// TIA Portal project "Quizshow" (V20)

(* hardware
DEVICE "S7-300/ET200M-Station_1"  S7-300 station
   slot 0: "Profilschiene_0"  Rail  6ES7 390-1***0-0AA0
   slot 2: "PLC_1"  CPU 315-2 PN/DP  6ES7 315-2EH14-0AB0  V3.2.18
      slot 2: "PROFINET-Schnittstelle_1"  PN-IO
         slot 1: "Port_1"  Port
         slot 2: "Port_2"  Port
   slot 4: "DI 16x24VDC_1"  DI16 x 24VDC, interrupt  6ES7 321-7BH01-0AB0
   slot 5: "DO 8x24VDC/0.5A_1"  DO8 x 24VDC / 0.5A  6ES7 322-8BF00-0AB0
*)

// ===== PLC "PLC_1"  CPU 315-2 PN/DP =====

VAR_GLOBAL   // PLC tag table "Standard-Variablentabelle"
   "Teilnehmer_1" AT %E0.0 : Bool;
   "Teilnehmer_2" AT %E0.1 : Bool;
   "TN_1-Lampe" AT %A0.0 : Bool;
   "TN_2-Lampe" AT %A0.1 : Bool;
   "TN_2-Gedrückt" AT %M0.1 : Bool;
   "TN_1-Gedrückt" AT %M0.0 : Bool;
   "Start-Taster" AT %E1.0 : Bool;
   "Freigabe erteilt" AT %A0.7 : Bool;
   "TN_3-Lampe" AT %A0.2 : Bool;
   "TN_4-Lampe" AT %A0.3 : Bool;
   "Teilnehmer_3" AT %E0.2 : Bool;
   "Teilnehmer_4" AT %E0.3 : Bool;
   "TN_3-Gedrückt" AT %M0.2 : Bool;
   "TN_4-Gedrückt" AT %M0.3 : Bool;
END_VAR

DATA_BLOCK "Quizshow_DB"   // DB1
{ S7_Optimized_Access := 'FALSE' }
VERSION : 0.1
// stored: InstanceOfName Quizshow
"Quizshow"
BEGIN
END_DATA_BLOCK

FUNCTION_BLOCK "Quizshow"   // FB6, FBD
{ S7_Optimized_Access := 'FALSE' }
VERSION : 0.1
BEGIN

REGION Network 1: Buzzer-Teilnehmer 1
   // Siehe Netzwerk 4.
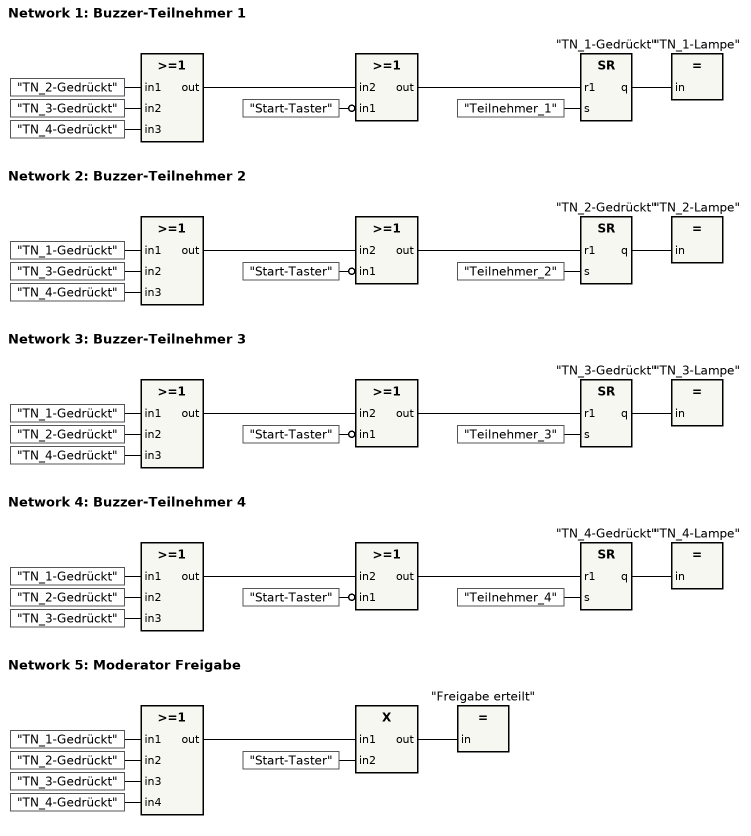
   IF "Teilnehmer_1" THEN
       "TN_1-Gedrückt" := TRUE;   // SR flip-flop
   END_IF;
   IF "TN_2-Gedrückt" OR "TN_3-Gedrückt" OR "TN_4-Gedrückt" OR NOT "Start-Taster" THEN
       "TN_1-Gedrückt" := FALSE;
   END_IF;
   "TN_1-Lampe" := "TN_1-Gedrückt";
END_REGION

REGION Network 2: Buzzer-Teilnehmer 2
   // Siehe Netzwerk 4.
   IF "Teilnehmer_2" THEN
       "TN_2-Gedrückt" := TRUE;   // SR flip-flop
   END_IF;
   IF "TN_1-Gedrückt" OR "TN_3-Gedrückt" OR "TN_4-Gedrückt" OR NOT "Start-Taster" THEN
       "TN_2-Gedrückt" := FALSE;
   END_IF;
   "TN_2-Lampe" := "TN_2-Gedrückt";
END_REGION

REGION Network 3: Buzzer-Teilnehmer 3
   // Siehe Netzwerk 4.
   IF "Teilnehmer_3" THEN
       "TN_3-Gedrückt" := TRUE;   // SR flip-flop
   END_IF;
   IF "TN_1-Gedrückt" OR "TN_2-Gedrückt" OR "TN_4-Gedrückt" OR NOT "Start-Taster" THEN
       "TN_3-Gedrückt" := FALSE;
   END_IF;
   "TN_3-Lampe" := "TN_3-Gedrückt";
END_REGION

REGION Network 4: Buzzer-Teilnehmer 4
   // Sobald der Moderator die Buzzer freigibt, und dieser Teilnehmer seinen Buzzer betätigt, geht seine Lampe an. Durch den SR-Flip Flop wird der Buzzer von diesem Teilnehmer durch den Moderator / die anderen Teilnehmer gesperrt, sodass dieser dann nicht buzzern kann.
   IF "Teilnehmer_4" THEN
       "TN_4-Gedrückt" := TRUE;   // SR flip-flop
   END_IF;
   IF "TN_1-Gedrückt" OR "TN_2-Gedrückt" OR "TN_3-Gedrückt" OR NOT "Start-Taster" THEN
       "TN_4-Gedrückt" := FALSE;
   END_IF;
   "TN_4-Lampe" := "TN_4-Gedrückt";
END_REGION

REGION Network 5: Moderator Freigabe
   // Der Moderator kann die Buzzer der Teilnehmer durch seinen Start-Taster freigeben. Dadurch leuchtet dann seine Lampe. Sobald nun ein Teilnehmer seinen Buzzer betätigt, wird das leuchten der Moderator-Lampe beendet.
   "Freigabe erteilt" := ("TN_1-Gedrückt" OR "TN_2-Gedrückt" OR "TN_3-Gedrückt" OR "TN_4-Gedrückt") XOR "Start-Taster";
END_REGION
END_FUNCTION_BLOCK

ORGANIZATION_BLOCK "Main"   // OB1, FBD
TITLE = "Main Program Sweep (Cycle)"
{ S7_Optimized_Access := 'FALSE' }
VERSION : 0.1
   VAR_TEMP
      OB1_EV_CLASS : Byte;   // Bits 0-3 = 1 (Coming event), Bits 4-7 = 1 (Event class 1)
      OB1_SCAN_1 : Byte;   // 1 (Cold restart scan 1 of OB 1), 3 (Scan 2-n of OB 1)
      OB1_PRIORITY : Byte;   // Priority of OB Execution
      OB1_OB_NUMBR : Byte;   // 1 (Organization block 1, OB1)
      OB1_RESERVED_1 : Byte;   // Reserved for system
      OB1_RESERVED_2 : Byte;   // Reserved for system
      OB1_PREV_CYCLE : Int;   // Cycle time of previous OB1 scan (milliseconds)
      OB1_MIN_CYCLE : Int;   // Minimum cycle time of OB1 (milliseconds)
      OB1_MAX_CYCLE : Int;   // Maximum cycle time of OB1 (milliseconds)
      OB1_DATE_TIME : Date_And_Time;   // Date and time OB1 started
   END_VAR
BEGIN

REGION Network 1
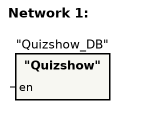
   "Quizshow_DB"();   // "Quizshow"
END_REGION
END_ORGANIZATION_BLOCK